PROGRAM SortTest
VAR
	TestArray0 : ARRAY[0..20] OF REAL := [
		1, 2, 3, 4, 5, 6, 7, 8, 9, 10,
		42, 3.14, 0.618, 1.618, 2.618
	];
	TestArray1 : ARRAY[0..3] OF STRING := ['aaa', 'g', 'aab', 'a'];
	
	sort_array : ARRAY[0..3] OF ST_TestStruct;	// TestArray2
	
	init : BOOL := TRUE;
	startSort : BOOL;
	
	order	: E_Order;
END_VAR


IF init THEN

	init := FALSE;

	reinit();
END_IF

IF startSort THEN

	startSort := FALSE;

	Sort(TestArray0, TestArray0[0], TestArray0[0], order);
	Sort(TestArray1, TestArray1[0], TestArray1[0], order);

	Sort(sort_array, sort_array[0], sort_array[0].by_this.nested_variable, order);
END_IF


METHOD reinit : BOOL
VAR_INPUT
END_VAR
VAR CONSTANT
	Array0 : ARRAY[0..20] OF REAL := [
		1, 2, 3, 4, 5, 6, 7, 8, 9, 10,
		42, 3.14, 0.618, 1.618, 2.618
	];
	Array1 : ARRAY[0..3] OF STRING := ['aaa', 'g', 'aab', 'a'];
END_VAR

TestArray0 := Array0;
TestArray1 := Array1;

sort_array[0].by_this.nested_variable := T#5S;
sort_array[1].by_this.nested_variable := T#1S;
sort_array[2].by_this.nested_variable := T#18D;
sort_array[3].by_this.nested_variable := T#42MS;
END_METHOD

END_PROGRAM

(* stored: Version 1.1.0.1, ProductVersion 3.1.4024.11
   POU SortTest: Id {d95a2e8d-bb47-456d-9afc-02b8a43bc324}, SpecialFunc None
   Method reinit: Id {d7862d1f-daa0-432e-8027-3852550d7ae0} *)
